Staubli VAL3: clkAirexOff.pgx

program clkAirexOff()
  local num idx
begin
  for idx = 0 to 5
    if statusValves[airexValve[idx]] == 1
      call toggleValve(airexValve[idx])
    endIf
  endFor
end
